TYPE ST1_ChangeBoxInfo :
STRUCT
	CheckedChangeBox		:	BOOL;
	ChangeBox 				:	ST0_ChangeBoxesInfo;
	HandShake				:  	st_HandshakeBase;
END_STRUCT
END_TYPE

(* stored: Version 1.1.0.1, ProductVersion 3.1.4024.13
   DUT ST1_ChangeBoxInfo: Id {5827aee1-069a-4ae1-81cb-1b14c525e54f} *)
